TYPE In_16_To_PLC :
STRUCT
	In AT %Q*:ARRAY [1..16] OF BOOL;
END_STRUCT
END_TYPE

(* stored: Version 1.1.0.1, ProductVersion 3.1.4024.15
   DUT In_16_To_PLC: Id {69491765-0113-47ce-a89d-11a73e999a42} *)
